FUNCTION "weight" : VOID	// FC 114
AUTHOR : gaw-be
FAMILY : temperat
NAME : display
VERSION : 0.1
BEGIN
// (block stored without names or comments; labels and parameter names are numbered)
NETWORK
TITLE =
      BLD   5;
      T     LD 10;
      TAK;
      T     LD 14;
      L     P##PARAM11;
      LAR1;
      L     W [AR1,P#0.0];
      T     LW 8;
      OPN   DB [LW 8];
      L     D [AR1,P#2.0];
      LAR1;
      L     LD 14;
      L     LD 10;
      L     W [AR1,P#34.0];
      L     -1;
      ==I;
      BLD   5;
      T     LD 10;
      TAK;
      T     LD 14;
      L     P##PARAM11;
      LAR1;
      L     W [AR1,P#0.0];
      T     LW 8;
      OPN   DB [LW 8];
      L     D [AR1,P#2.0];
      LAR1;
      L     LD 14;
      L     LD 10;
      R      [AR1,P#36.0];
      L     #PARAM2;
      BLD   5;
      T     LD 10;
      TAK;
      T     LD 14;
      L     P##PARAM11;
      LAR1;
      L     W [AR1,P#0.0];
      T     LW 8;
      OPN   DB [LW 8];
      L     D [AR1,P#2.0];
      LAR1;
      L     LD 14;
      L     LD 10;
      L     W [AR1,P#34.0];
      <>I;
      JC    M006;
      BLD   5;
      T     LD 10;
      TAK;
      T     LD 14;
      L     P##PARAM11;
      LAR1;
      L     W [AR1,P#0.0];
      T     LW 8;
      OPN   DB [LW 8];
      L     D [AR1,P#2.0];
      LAR1;
      L     LD 14;
      L     LD 10;
      A      [AR1,P#36.0];
      JC    M001;
      BLD   5;
      T     LD 10;
      TAK;
      T     LD 14;
      L     P##PARAM10;
      LAR1;
      L     W [AR1,P#0.0];
      T     LW 8;
      OPN   DB [LW 8];
      L     D [AR1,P#2.0];
      LAR1;
      L     LD 14;
      L     LD 10;
      L     B [AR1,P#4.0];
      BLD   5;
      T     LD 10;
      TAK;
      T     LD 14;
      L     P##PARAM11;
      LAR1;
      L     W [AR1,P#0.0];
      T     LW 8;
      OPN   DB [LW 8];
      L     D [AR1,P#2.0];
      LAR1;
      L     LD 14;
      L     LD 10;
      T     B [AR1,P#4.0];
      BLD   5;
      T     LD 10;
      TAK;
      T     LD 14;
      L     P##PARAM10;
      LAR1;
      L     W [AR1,P#0.0];
      T     LW 8;
      OPN   DB [LW 8];
      L     D [AR1,P#2.0];
      LAR1;
      L     LD 14;
      L     LD 10;
      L     D [AR1,P#6.0];
      BLD   5;
      T     LD 10;
      TAK;
      T     LD 14;
      L     P##PARAM11;
      LAR1;
      L     W [AR1,P#0.0];
      T     LW 8;
      OPN   DB [LW 8];
      L     D [AR1,P#2.0];
      LAR1;
      L     LD 14;
      L     LD 10;
      T     D [AR1,P#6.0];
      BLD   5;
      T     LD 10;
      TAK;
      T     LD 14;
      L     P##PARAM10;
      LAR1;
      L     W [AR1,P#0.0];
      T     LW 8;
      OPN   DB [LW 8];
      L     D [AR1,P#2.0];
      LAR1;
      L     LD 14;
      L     LD 10;
      L     D [AR1,P#10.0];
      BLD   5;
      T     LD 10;
      TAK;
      T     LD 14;
      L     P##PARAM11;
      LAR1;
      L     W [AR1,P#0.0];
      T     LW 8;
      OPN   DB [LW 8];
      L     D [AR1,P#2.0];
      LAR1;
      L     LD 14;
      L     LD 10;
      T     D [AR1,P#10.0];
      BLD   5;
      T     LD 10;
      TAK;
      T     LD 14;
      L     P##PARAM10;
      LAR1;
      L     W [AR1,P#0.0];
      T     LW 8;
      OPN   DB [LW 8];
      L     D [AR1,P#2.0];
      LAR1;
      L     LD 14;
      L     LD 10;
      L     D [AR1,P#14.0];
      BLD   5;
      T     LD 10;
      TAK;
      T     LD 14;
      L     P##PARAM11;
      LAR1;
      L     W [AR1,P#0.0];
      T     LW 8;
      OPN   DB [LW 8];
      L     D [AR1,P#2.0];
      LAR1;
      L     LD 14;
      L     LD 10;
      T     D [AR1,P#14.0];
      BLD   5;
      T     LD 10;
      TAK;
      T     LD 14;
      L     P##PARAM10;
      LAR1;
      L     W [AR1,P#0.0];
      T     LW 8;
      OPN   DB [LW 8];
      L     D [AR1,P#2.0];
      LAR1;
      L     LD 14;
      L     LD 10;
      L     D [AR1,P#18.0];
      BLD   5;
      T     LD 10;
      TAK;
      T     LD 14;
      L     P##PARAM11;
      LAR1;
      L     W [AR1,P#0.0];
      T     LW 8;
      OPN   DB [LW 8];
      L     D [AR1,P#2.0];
      LAR1;
      L     LD 14;
      L     LD 10;
      T     D [AR1,P#18.0];
      BLD   5;
      T     LD 10;
      TAK;
      T     LD 14;
      L     P##PARAM10;
      LAR1;
      L     W [AR1,P#0.0];
      T     LW 8;
      OPN   DB [LW 8];
      L     D [AR1,P#2.0];
      LAR1;
      L     LD 14;
      L     LD 10;
      L     D [AR1,P#22.0];
      BLD   5;
      T     LD 10;
      TAK;
      T     LD 14;
      L     P##PARAM11;
      LAR1;
      L     W [AR1,P#0.0];
      T     LW 8;
      OPN   DB [LW 8];
      L     D [AR1,P#2.0];
      LAR1;
      L     LD 14;
      L     LD 10;
      T     D [AR1,P#22.0];
      BLD   5;
      T     LD 10;
      TAK;
      T     LD 14;
      L     P##PARAM10;
      LAR1;
      L     W [AR1,P#0.0];
      T     LW 8;
      OPN   DB [LW 8];
      L     D [AR1,P#2.0];
      LAR1;
      L     LD 14;
      L     LD 10;
      L     D [AR1,P#26.0];
      BLD   5;
      T     LD 10;
      TAK;
      T     LD 14;
      L     P##PARAM11;
      LAR1;
      L     W [AR1,P#0.0];
      T     LW 8;
      OPN   DB [LW 8];
      L     D [AR1,P#2.0];
      LAR1;
      L     LD 14;
      L     LD 10;
      T     D [AR1,P#26.0];
      BLD   5;
      T     LD 10;
      TAK;
      T     LD 14;
      L     P##PARAM10;
      LAR1;
      L     W [AR1,P#0.0];
      T     LW 8;
      OPN   DB [LW 8];
      L     D [AR1,P#2.0];
      LAR1;
      L     LD 14;
      L     LD 10;
      L     D [AR1,P#30.0];
      BLD   5;
      T     LD 10;
      TAK;
      T     LD 14;
      L     P##PARAM11;
      LAR1;
      L     W [AR1,P#0.0];
      T     LW 8;
      OPN   DB [LW 8];
      L     D [AR1,P#2.0];
      LAR1;
      L     LD 14;
      L     LD 10;
      T     D [AR1,P#30.0];
      SET;
      BLD   5;
      T     LD 10;
      TAK;
      T     LD 14;
      L     P##PARAM11;
      LAR1;
      L     W [AR1,P#0.0];
      T     LW 8;
      OPN   DB [LW 8];
      L     D [AR1,P#2.0];
      LAR1;
      L     LD 14;
      L     LD 10;
      =      [AR1,P#36.0];
M001: BLD   5;
      T     LD 10;
      TAK;
      T     LD 14;
      L     P##PARAM10;
      LAR1;
      L     W [AR1,P#0.0];
      T     LW 8;
      OPN   DB [LW 8];
      L     D [AR1,P#2.0];
      LAR1;
      L     LD 14;
      L     LD 10;
      L     D [AR1,P#0.0];
      BLD   5;
      T     LD 10;
      TAK;
      T     LD 14;
      L     P##PARAM11;
      LAR1;
      L     W [AR1,P#0.0];
      T     LW 8;
      OPN   DB [LW 8];
      L     D [AR1,P#2.0];
      LAR1;
      L     LD 14;
      L     LD 10;
      T     D [AR1,P#0.0];
      BLD   5;
      T     LD 10;
      TAK;
      T     LD 14;
      L     P##PARAM11;
      LAR1;
      L     W [AR1,P#0.0];
      T     LW 8;
      OPN   DB [LW 8];
      L     D [AR1,P#2.0];
      LAR1;
      L     LD 14;
      L     LD 10;
      L     B [AR1,P#4.0];
      BLD   5;
      T     LD 10;
      TAK;
      T     LD 14;
      L     P##PARAM10;
      LAR1;
      L     W [AR1,P#0.0];
      T     LW 8;
      OPN   DB [LW 8];
      L     D [AR1,P#2.0];
      LAR1;
      L     LD 14;
      L     LD 10;
      T     B [AR1,P#4.0];
      BLD   5;
      T     LD 10;
      TAK;
      T     LD 14;
      L     P##PARAM11;
      LAR1;
      L     W [AR1,P#0.0];
      T     LW 8;
      OPN   DB [LW 8];
      L     D [AR1,P#2.0];
      LAR1;
      L     LD 14;
      L     LD 10;
      L     D [AR1,P#6.0];
      BLD   5;
      T     LD 10;
      TAK;
      T     LD 14;
      L     P##PARAM10;
      LAR1;
      L     W [AR1,P#0.0];
      T     LW 8;
      OPN   DB [LW 8];
      L     D [AR1,P#2.0];
      LAR1;
      L     LD 14;
      L     LD 10;
      T     D [AR1,P#6.0];
      BLD   5;
      T     LD 10;
      TAK;
      T     LD 14;
      L     P##PARAM11;
      LAR1;
      L     W [AR1,P#0.0];
      T     LW 8;
      OPN   DB [LW 8];
      L     D [AR1,P#2.0];
      LAR1;
      L     LD 14;
      L     LD 10;
      L     D [AR1,P#10.0];
      BLD   5;
      T     LD 10;
      TAK;
      T     LD 14;
      L     P##PARAM10;
      LAR1;
      L     W [AR1,P#0.0];
      T     LW 8;
      OPN   DB [LW 8];
      L     D [AR1,P#2.0];
      LAR1;
      L     LD 14;
      L     LD 10;
      T     D [AR1,P#10.0];
      BLD   5;
      T     LD 10;
      TAK;
      T     LD 14;
      L     P##PARAM11;
      LAR1;
      L     W [AR1,P#0.0];
      T     LW 8;
      OPN   DB [LW 8];
      L     D [AR1,P#2.0];
      LAR1;
      L     LD 14;
      L     LD 10;
      L     D [AR1,P#14.0];
      BLD   5;
      T     LD 10;
      TAK;
      T     LD 14;
      L     P##PARAM10;
      LAR1;
      L     W [AR1,P#0.0];
      T     LW 8;
      OPN   DB [LW 8];
      L     D [AR1,P#2.0];
      LAR1;
      L     LD 14;
      L     LD 10;
      T     D [AR1,P#14.0];
      BLD   5;
      T     LD 10;
      TAK;
      T     LD 14;
      L     P##PARAM11;
      LAR1;
      L     W [AR1,P#0.0];
      T     LW 8;
      OPN   DB [LW 8];
      L     D [AR1,P#2.0];
      LAR1;
      L     LD 14;
      L     LD 10;
      L     D [AR1,P#26.0];
      BLD   5;
      T     LD 10;
      TAK;
      T     LD 14;
      L     P##PARAM11;
      LAR1;
      L     W [AR1,P#0.0];
      T     LW 8;
      OPN   DB [LW 8];
      L     D [AR1,P#2.0];
      LAR1;
      L     LD 14;
      L     LD 10;
      L     D [AR1,P#30.0];
      >R;
      JC    M002;
      BLD   5;
      T     LD 10;
      TAK;
      T     LD 14;
      L     P##PARAM11;
      LAR1;
      L     W [AR1,P#0.0];
      T     LW 8;
      OPN   DB [LW 8];
      L     D [AR1,P#2.0];
      LAR1;
      L     LD 14;
      L     LD 10;
      L     D [AR1,P#26.0];
      BLD   5;
      T     LD 10;
      TAK;
      T     LD 14;
      L     P##PARAM11;
      LAR1;
      L     W [AR1,P#0.0];
      T     LW 8;
      OPN   DB [LW 8];
      L     D [AR1,P#2.0];
      LAR1;
      L     LD 14;
      L     LD 10;
      L     D [AR1,P#22.0];
      <R;
      JC    M002;
      BLD   5;
      T     LD 10;
      TAK;
      T     LD 14;
      L     P##PARAM11;
      LAR1;
      L     W [AR1,P#0.0];
      T     LW 8;
      OPN   DB [LW 8];
      L     D [AR1,P#2.0];
      LAR1;
      L     LD 14;
      L     LD 10;
      L     D [AR1,P#26.0];
M002: BLD   5;
      T     LD 10;
      TAK;
      T     LD 14;
      L     P##PARAM11;
      LAR1;
      L     W [AR1,P#0.0];
      T     LW 8;
      OPN   DB [LW 8];
      L     D [AR1,P#2.0];
      LAR1;
      L     LD 14;
      L     LD 10;
      T     D [AR1,P#26.0];
      BLD   5;
      T     LD 10;
      TAK;
      T     LD 14;
      L     P##PARAM11;
      LAR1;
      L     W [AR1,P#0.0];
      T     LW 8;
      OPN   DB [LW 8];
      L     D [AR1,P#2.0];
      LAR1;
      L     LD 14;
      L     LD 10;
      L     D [AR1,P#26.0];
      BLD   5;
      T     LD 10;
      TAK;
      T     LD 14;
      L     P##PARAM10;
      LAR1;
      L     W [AR1,P#0.0];
      T     LW 8;
      OPN   DB [LW 8];
      L     D [AR1,P#2.0];
      LAR1;
      L     LD 14;
      L     LD 10;
      T     D [AR1,P#26.0];
      BLD   5;
      T     LD 10;
      TAK;
      T     LD 14;
      L     P##PARAM11;
      LAR1;
      L     W [AR1,P#0.0];
      T     LW 8;
      OPN   DB [LW 8];
      L     D [AR1,P#2.0];
      LAR1;
      L     LD 14;
      L     LD 10;
      L     D [AR1,P#30.0];
      BLD   5;
      T     LD 10;
      TAK;
      T     LD 14;
      L     P##PARAM11;
      LAR1;
      L     W [AR1,P#0.0];
      T     LW 8;
      OPN   DB [LW 8];
      L     D [AR1,P#2.0];
      LAR1;
      L     LD 14;
      L     LD 10;
      L     D [AR1,P#14.0];
      >R;
      JC    M003;
      BLD   5;
      T     LD 10;
      TAK;
      T     LD 14;
      L     P##PARAM11;
      LAR1;
      L     W [AR1,P#0.0];
      T     LW 8;
      OPN   DB [LW 8];
      L     D [AR1,P#2.0];
      LAR1;
      L     LD 14;
      L     LD 10;
      L     D [AR1,P#30.0];
      BLD   5;
      T     LD 10;
      TAK;
      T     LD 14;
      L     P##PARAM11;
      LAR1;
      L     W [AR1,P#0.0];
      T     LW 8;
      OPN   DB [LW 8];
      L     D [AR1,P#2.0];
      LAR1;
      L     LD 14;
      L     LD 10;
      L     D [AR1,P#26.0];
      <R;
      JC    M003;
      BLD   5;
      T     LD 10;
      TAK;
      T     LD 14;
      L     P##PARAM11;
      LAR1;
      L     W [AR1,P#0.0];
      T     LW 8;
      OPN   DB [LW 8];
      L     D [AR1,P#2.0];
      LAR1;
      L     LD 14;
      L     LD 10;
      L     D [AR1,P#30.0];
M003: BLD   5;
      T     LD 10;
      TAK;
      T     LD 14;
      L     P##PARAM11;
      LAR1;
      L     W [AR1,P#0.0];
      T     LW 8;
      OPN   DB [LW 8];
      L     D [AR1,P#2.0];
      LAR1;
      L     LD 14;
      L     LD 10;
      T     D [AR1,P#30.0];
      BLD   5;
      T     LD 10;
      TAK;
      T     LD 14;
      L     P##PARAM11;
      LAR1;
      L     W [AR1,P#0.0];
      T     LW 8;
      OPN   DB [LW 8];
      L     D [AR1,P#2.0];
      LAR1;
      L     LD 14;
      L     LD 10;
      L     D [AR1,P#30.0];
      BLD   5;
      T     LD 10;
      TAK;
      T     LD 14;
      L     P##PARAM10;
      LAR1;
      L     W [AR1,P#0.0];
      T     LW 8;
      OPN   DB [LW 8];
      L     D [AR1,P#2.0];
      LAR1;
      L     LD 14;
      L     LD 10;
      T     D [AR1,P#30.0];
      BLD   5;
      T     LD 10;
      TAK;
      T     LD 14;
      L     P##PARAM11;
      LAR1;
      L     W [AR1,P#0.0];
      T     LW 8;
      OPN   DB [LW 8];
      L     D [AR1,P#2.0];
      LAR1;
      L     LD 14;
      L     LD 10;
      L     D [AR1,P#22.0];
      BLD   5;
      T     LD 10;
      TAK;
      T     LD 14;
      L     P##PARAM11;
      LAR1;
      L     W [AR1,P#0.0];
      T     LW 8;
      OPN   DB [LW 8];
      L     D [AR1,P#2.0];
      LAR1;
      L     LD 14;
      L     LD 10;
      L     D [AR1,P#26.0];
      >R;
      JC    M004;
      BLD   5;
      T     LD 10;
      TAK;
      T     LD 14;
      L     P##PARAM11;
      LAR1;
      L     W [AR1,P#0.0];
      T     LW 8;
      OPN   DB [LW 8];
      L     D [AR1,P#2.0];
      LAR1;
      L     LD 14;
      L     LD 10;
      L     D [AR1,P#22.0];
      BLD   5;
      T     LD 10;
      TAK;
      T     LD 14;
      L     P##PARAM11;
      LAR1;
      L     W [AR1,P#0.0];
      T     LW 8;
      OPN   DB [LW 8];
      L     D [AR1,P#2.0];
      LAR1;
      L     LD 14;
      L     LD 10;
      L     D [AR1,P#18.0];
      <R;
      JC    M004;
      BLD   5;
      T     LD 10;
      TAK;
      T     LD 14;
      L     P##PARAM11;
      LAR1;
      L     W [AR1,P#0.0];
      T     LW 8;
      OPN   DB [LW 8];
      L     D [AR1,P#2.0];
      LAR1;
      L     LD 14;
      L     LD 10;
      L     D [AR1,P#22.0];
M004: BLD   5;
      T     LD 10;
      TAK;
      T     LD 14;
      L     P##PARAM11;
      LAR1;
      L     W [AR1,P#0.0];
      T     LW 8;
      OPN   DB [LW 8];
      L     D [AR1,P#2.0];
      LAR1;
      L     LD 14;
      L     LD 10;
      T     D [AR1,P#22.0];
      BLD   5;
      T     LD 10;
      TAK;
      T     LD 14;
      L     P##PARAM11;
      LAR1;
      L     W [AR1,P#0.0];
      T     LW 8;
      OPN   DB [LW 8];
      L     D [AR1,P#2.0];
      LAR1;
      L     LD 14;
      L     LD 10;
      L     D [AR1,P#22.0];
      BLD   5;
      T     LD 10;
      TAK;
      T     LD 14;
      L     P##PARAM10;
      LAR1;
      L     W [AR1,P#0.0];
      T     LW 8;
      OPN   DB [LW 8];
      L     D [AR1,P#2.0];
      LAR1;
      L     LD 14;
      L     LD 10;
      T     D [AR1,P#22.0];
      BLD   5;
      T     LD 10;
      TAK;
      T     LD 14;
      L     P##PARAM11;
      LAR1;
      L     W [AR1,P#0.0];
      T     LW 8;
      OPN   DB [LW 8];
      L     D [AR1,P#2.0];
      LAR1;
      L     LD 14;
      L     LD 10;
      L     D [AR1,P#18.0];
      BLD   5;
      T     LD 10;
      TAK;
      T     LD 14;
      L     P##PARAM11;
      LAR1;
      L     W [AR1,P#0.0];
      T     LW 8;
      OPN   DB [LW 8];
      L     D [AR1,P#2.0];
      LAR1;
      L     LD 14;
      L     LD 10;
      L     D [AR1,P#22.0];
      >R;
      JC    M005;
      BLD   5;
      T     LD 10;
      TAK;
      T     LD 14;
      L     P##PARAM11;
      LAR1;
      L     W [AR1,P#0.0];
      T     LW 8;
      OPN   DB [LW 8];
      L     D [AR1,P#2.0];
      LAR1;
      L     LD 14;
      L     LD 10;
      L     D [AR1,P#18.0];
      BLD   5;
      T     LD 10;
      TAK;
      T     LD 14;
      L     P##PARAM11;
      LAR1;
      L     W [AR1,P#0.0];
      T     LW 8;
      OPN   DB [LW 8];
      L     D [AR1,P#2.0];
      LAR1;
      L     LD 14;
      L     LD 10;
      L     D [AR1,P#10.0];
      <R;
      JC    M005;
      BLD   5;
      T     LD 10;
      TAK;
      T     LD 14;
      L     P##PARAM11;
      LAR1;
      L     W [AR1,P#0.0];
      T     LW 8;
      OPN   DB [LW 8];
      L     D [AR1,P#2.0];
      LAR1;
      L     LD 14;
      L     LD 10;
      L     D [AR1,P#18.0];
M005: BLD   5;
      T     LD 10;
      TAK;
      T     LD 14;
      L     P##PARAM11;
      LAR1;
      L     W [AR1,P#0.0];
      T     LW 8;
      OPN   DB [LW 8];
      L     D [AR1,P#2.0];
      LAR1;
      L     LD 14;
      L     LD 10;
      T     D [AR1,P#18.0];
      BLD   5;
      T     LD 10;
      TAK;
      T     LD 14;
      L     P##PARAM11;
      LAR1;
      L     W [AR1,P#0.0];
      T     LW 8;
      OPN   DB [LW 8];
      L     D [AR1,P#2.0];
      LAR1;
      L     LD 14;
      L     LD 10;
      L     D [AR1,P#18.0];
      BLD   5;
      T     LD 10;
      TAK;
      T     LD 14;
      L     P##PARAM10;
      LAR1;
      L     W [AR1,P#0.0];
      T     LW 8;
      OPN   DB [LW 8];
      L     D [AR1,P#2.0];
      LAR1;
      L     LD 14;
      L     LD 10;
      T     D [AR1,P#18.0];
M006: NOP   0;
NETWORK
TITLE =
      L     #PARAM1;
      T     #PARAM8;
      T     LD 0;
      BLD   5;
      T     LD 10;
      TAK;
      T     LD 14;
      L     P##PARAM10;
      LAR1;
      L     W [AR1,P#0.0];
      T     LW 8;
      OPN   DB [LW 8];
      L     D [AR1,P#2.0];
      LAR1;
      L     LD 14;
      L     LD 10;
      L     D [AR1,P#14.0];
      BLD   5;
      T     LD 10;
      TAK;
      T     LD 14;
      L     P##PARAM10;
      LAR1;
      L     W [AR1,P#0.0];
      T     LW 8;
      OPN   DB [LW 8];
      L     D [AR1,P#2.0];
      LAR1;
      L     LD 14;
      L     LD 10;
      L     D [AR1,P#10.0];
      -R;
      L     LD 0;
      *R;
      L     1.000000e+02;
      /R;
      BLD   5;
      T     LD 10;
      TAK;
      T     LD 14;
      L     P##PARAM10;
      LAR1;
      L     W [AR1,P#0.0];
      T     LW 8;
      OPN   DB [LW 8];
      L     D [AR1,P#2.0];
      LAR1;
      L     LD 14;
      L     LD 10;
      L     D [AR1,P#10.0];
      +R;
      T     #PARAM9;
      T     LD 4;
      BLD   5;
      T     LD 10;
      TAK;
      T     LD 14;
      L     P##PARAM10;
      LAR1;
      L     W [AR1,P#0.0];
      T     LW 8;
      OPN   DB [LW 8];
      L     D [AR1,P#2.0];
      LAR1;
      L     LD 14;
      L     LD 10;
      L     B [AR1,P#4.0];
      L     0;
      ==I;
      JC    M007;
      BLD   5;
      T     LD 10;
      TAK;
      T     LD 14;
      L     P##PARAM10;
      LAR1;
      L     W [AR1,P#0.0];
      T     LW 8;
      OPN   DB [LW 8];
      L     D [AR1,P#2.0];
      LAR1;
      L     LD 14;
      L     LD 10;
      L     B [AR1,P#4.0];
      L     1;
      ==I;
      JC    M008;
      L     -1.000000e+02;
      JU    M009;
M007: L     LD 0;
      JU    M009;
M008: L     LD 4;
M009: BLD   5;
      T     LD 10;
      TAK;
      T     LD 14;
      L     P##PARAM10;
      LAR1;
      L     W [AR1,P#0.0];
      T     LW 8;
      OPN   DB [LW 8];
      L     D [AR1,P#2.0];
      LAR1;
      L     LD 14;
      L     LD 10;
      T     D [AR1,P#0.0];
NETWORK
TITLE =
      BLD   5;
      T     LD 10;
      TAK;
      T     LD 14;
      L     P##PARAM10;
      LAR1;
      L     W [AR1,P#0.0];
      T     LW 8;
      OPN   DB [LW 8];
      L     D [AR1,P#2.0];
      LAR1;
      L     LD 14;
      L     LD 10;
      L     D [AR1,P#18.0];
      L     LD 4;
      >=R;
      S     #PARAM7;
      BLD   5;
      T     LD 10;
      TAK;
      T     LD 14;
      L     P##PARAM10;
      LAR1;
      L     W [AR1,P#0.0];
      T     LW 8;
      OPN   DB [LW 8];
      L     D [AR1,P#2.0];
      LAR1;
      L     LD 14;
      L     LD 10;
      L     D [AR1,P#18.0];
      BLD   5;
      T     LD 10;
      TAK;
      T     LD 14;
      L     P##PARAM10;
      LAR1;
      L     W [AR1,P#0.0];
      T     LW 8;
      OPN   DB [LW 8];
      L     D [AR1,P#2.0];
      LAR1;
      L     LD 14;
      L     LD 10;
      L     D [AR1,P#6.0];
      +R;
      L     LD 4;
      <=R;
      R     #PARAM7;
      BLD   5;
      T     LD 10;
      TAK;
      T     LD 14;
      L     P##PARAM10;
      LAR1;
      L     W [AR1,P#0.0];
      T     LW 8;
      OPN   DB [LW 8];
      L     D [AR1,P#2.0];
      LAR1;
      L     LD 14;
      L     LD 10;
      L     D [AR1,P#22.0];
      L     LD 4;
      >=R;
      S     #PARAM6;
      BLD   5;
      T     LD 10;
      TAK;
      T     LD 14;
      L     P##PARAM10;
      LAR1;
      L     W [AR1,P#0.0];
      T     LW 8;
      OPN   DB [LW 8];
      L     D [AR1,P#2.0];
      LAR1;
      L     LD 14;
      L     LD 10;
      L     D [AR1,P#22.0];
      BLD   5;
      T     LD 10;
      TAK;
      T     LD 14;
      L     P##PARAM10;
      LAR1;
      L     W [AR1,P#0.0];
      T     LW 8;
      OPN   DB [LW 8];
      L     D [AR1,P#2.0];
      LAR1;
      L     LD 14;
      L     LD 10;
      L     D [AR1,P#6.0];
      +R;
      L     LD 4;
      <=R;
      R     #PARAM6;
      BLD   5;
      T     LD 10;
      TAK;
      T     LD 14;
      L     P##PARAM10;
      LAR1;
      L     W [AR1,P#0.0];
      T     LW 8;
      OPN   DB [LW 8];
      L     D [AR1,P#2.0];
      LAR1;
      L     LD 14;
      L     LD 10;
      L     D [AR1,P#26.0];
      L     LD 4;
      <=R;
      S     #PARAM5;
      BLD   5;
      T     LD 10;
      TAK;
      T     LD 14;
      L     P##PARAM10;
      LAR1;
      L     W [AR1,P#0.0];
      T     LW 8;
      OPN   DB [LW 8];
      L     D [AR1,P#2.0];
      LAR1;
      L     LD 14;
      L     LD 10;
      L     D [AR1,P#26.0];
      BLD   5;
      T     LD 10;
      TAK;
      T     LD 14;
      L     P##PARAM10;
      LAR1;
      L     W [AR1,P#0.0];
      T     LW 8;
      OPN   DB [LW 8];
      L     D [AR1,P#2.0];
      LAR1;
      L     LD 14;
      L     LD 10;
      L     D [AR1,P#6.0];
      -R;
      L     LD 4;
      >=R;
      R     #PARAM5;
      BLD   5;
      T     LD 10;
      TAK;
      T     LD 14;
      L     P##PARAM10;
      LAR1;
      L     W [AR1,P#0.0];
      T     LW 8;
      OPN   DB [LW 8];
      L     D [AR1,P#2.0];
      LAR1;
      L     LD 14;
      L     LD 10;
      L     D [AR1,P#30.0];
      L     LD 4;
      <=R;
      S     #PARAM4;
      BLD   5;
      T     LD 10;
      TAK;
      T     LD 14;
      L     P##PARAM10;
      LAR1;
      L     W [AR1,P#0.0];
      T     LW 8;
      OPN   DB [LW 8];
      L     D [AR1,P#2.0];
      LAR1;
      L     LD 14;
      L     LD 10;
      L     D [AR1,P#30.0];
      BLD   5;
      T     LD 10;
      TAK;
      T     LD 14;
      L     P##PARAM10;
      LAR1;
      L     W [AR1,P#0.0];
      T     LW 8;
      OPN   DB [LW 8];
      L     D [AR1,P#2.0];
      LAR1;
      L     LD 14;
      L     LD 10;
      L     D [AR1,P#6.0];
      -R;
      L     LD 4;
      >=R;
      R     #PARAM4;
      AN    #PARAM3;
      JC    M010;
      SET;
      =     #PARAM4;
      =     #PARAM7;
M010: NOP   0;
      BLD   5;
      T     LD 10;
      TAK;
      T     LD 14;
      L     P##PARAM10;
      LAR1;
      L     W [AR1,P#0.0];
      T     LW 8;
      OPN   DB [LW 8];
      L     D [AR1,P#2.0];
      LAR1;
      L     LD 14;
      L     LD 10;
      L     D [AR1,P#0.0];
      L     -1.000000e+02;
      <>R;
      JC    M011;
      SET;
      =     #PARAM4;
      =     #PARAM7;
M011: NOP   0;
END_FUNCTION

FUNCTION "ALARM_BLOCK" : VOID	// FC 115
AUTHOR : BAJZEK
FAMILY : ALARM
NAME : A_BLOCK
VERSION : 0.1
BEGIN
// (block stored without names or comments; labels and parameter names are numbered)
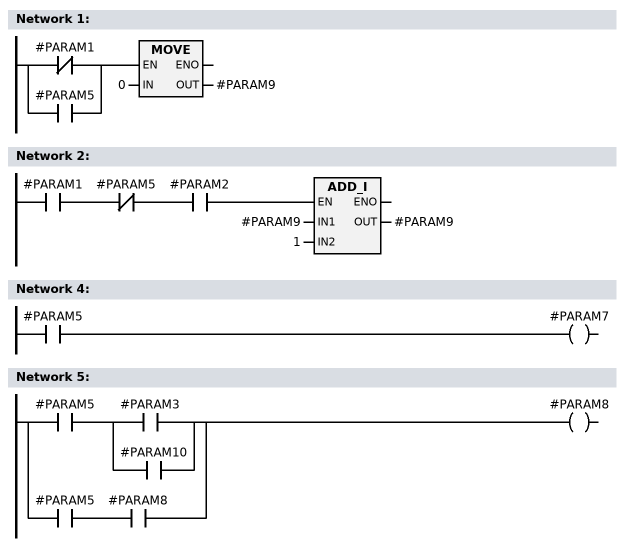
NETWORK
TITLE =
      A(;
      ON    #PARAM1;
      O     #PARAM5;
      );
      JNB   M001;
      L     0;
      T     #PARAM9;
M001: NOP   0;
NETWORK
TITLE =
      A     #PARAM1;
      AN    #PARAM5;
      A     #PARAM2;
      JNB   M002;
      L     #PARAM9;
      L     1;
      +I;
      T     #PARAM9;
M002: NOP   0;
NETWORK
TITLE =
      A(;
      A(;
      L     #PARAM9;
      L     #PARAM4;
      >=I;
      );
      S     #PARAM5;
      A     #PARAM6;
      AN    #PARAM1;
      R     #PARAM5;
      A     #PARAM5;
      );
      A     #PARAM10;
      S     #PARAM6;
      AN    #PARAM5;
      R     #PARAM6;
      NOP   0;
NETWORK
TITLE =
      A     #PARAM5;
      =     #PARAM7;
NETWORK
TITLE =
      A     #PARAM5;
      A(;
      O     #PARAM3;
      O     #PARAM10;
      );
      O;
      A     #PARAM5;
      A     #PARAM8;
      =     #PARAM8;
NETWORK
TITLE =
      CLR;
      =     #PARAM10;
END_FUNCTION

DATA_BLOCK "CLOCK_OP"	// DB 5
AUTHOR : gaw-be
FAMILY : GAW
NAME : UHR
VERSION : 0.1
BEGIN
// 24 bytes; values not shown
END_DATA_BLOCK

DATA_BLOCK "TransferValves"	// DB 10
AUTHOR : gaw-be
FAMILY : Valves
NAME : Data
VERSION : 0.1
BEGIN
// 16 bytes; values not shown
END_DATA_BLOCK

DATA_BLOCK "TransferMotor"	// DB 11
AUTHOR : gaw-be
FAMILY : Motor
NAME : Data
VERSION : 0.1
BEGIN
// 16 bytes; values not shown
END_DATA_BLOCK

DATA_BLOCK "TransferLevel"	// DB 12
AUTHOR : gaw-be
FAMILY : Level
NAME : Data
VERSION : 0.1
BEGIN
// 140 bytes; values not shown
END_DATA_BLOCK

DATA_BLOCK "TransferTemperature"	// DB 14
AUTHOR : gaw-be
FAMILY : Temp.
NAME : Data
VERSION : 0.1
BEGIN
// 72 bytes; values not shown
END_DATA_BLOCK

DATA_BLOCK "TransferWeight"	// DB 18
AUTHOR : gaw-be
FAMILY : Viskosit
NAME : Data
VERSION : 0.1
BEGIN
// 72 bytes; values not shown
END_DATA_BLOCK

DATA_BLOCK "TransferGenerell"	// DB 30
VERSION : 0.1
BEGIN
// 12 bytes; values not shown
END_DATA_BLOCK

DATA_BLOCK "TransferRecipe"	// DB 90
AUTHOR : gaw-be
FAMILY : Valves
NAME : Data
VERSION : 0.1
BEGIN
// 104 bytes; values not shown
END_DATA_BLOCK

DATA_BLOCK "TransferBatch"	// DB 91
AUTHOR : gaw-be
FAMILY : Valves
NAME : Data
VERSION : 0.1
BEGIN
// 104 bytes; values not shown
END_DATA_BLOCK

DATA_BLOCK "DataBatchControl"	// DB 92
VERSION : 0.0
"Batch"
BEGIN
END_DATA_BLOCK

DATA_BLOCK "ALARMTIME"	// DB 100
AUTHOR : BAJZEK
FAMILY : ALARM
NAME : ALTIME
VERSION : 0.1
BEGIN
// 288 bytes; values not shown
END_DATA_BLOCK

DATA_BLOCK "ALARMBLOCK"	// DB 110
AUTHOR : BAJZEK
FAMILY : ALARM
NAME : ALARM
VERSION : 0.1
BEGIN
// 18 bytes; values not shown
END_DATA_BLOCK

DATA_BLOCK "ALARM_ACK_OP"	// DB 115
AUTHOR : BAJZEK
FAMILY : ALARM
NAME : ALARM
VERSION : 0.1
BEGIN
// 18 bytes; values not shown
END_DATA_BLOCK

DATA_BLOCK "LAMPS_ACK"	// DB 120
AUTHOR : BAJZEK
FAMILY : ALARM
NAME : ALARM
VERSION : 0.1
BEGIN
// 18 bytes; values not shown
END_DATA_BLOCK

ORGANIZATION_BLOCK OB 1
VERSION : 0.1
BEGIN
// (block stored without names or comments; labels and parameter names are numbered)
NETWORK
TITLE =
      AN    "1_second";
      L     S5T#1S;
      SD    T 0;
      NOP   0;
      NOP   0;
      NOP   0;
      A     T 0;
      =     "1_second";
NETWORK
TITLE =
      A     "Signal_0";
      =     "PB_LAMP_ACK";
NETWORK
TITLE =
      A     DB5.DBX 21.2;
      FP    "LB_OP_PULS";
      L     S5T#1M;
      SF    T 4;
      NOP   0;
      NOP   0;
      NOP   0;
      A     T 4;
      =     "OP_COMM_OK";
NETWORK
TITLE =
      SET;
      R     "Signal_0";
      S     "Signal_1";
      L     LW 6;
      T     "Cycle_Time";
      UC    "CLOCK_FB";
      UC    "ALARM_HANDLING";
      UC    "ALARM";
      UC    "preparation";
      UC    "Devices";
      UC    "BatchControl";
END_ORGANIZATION_BLOCK
